KUKA KRL program: ab_com_01_st01_g01.src, ab_com_01_st01_g01.dat

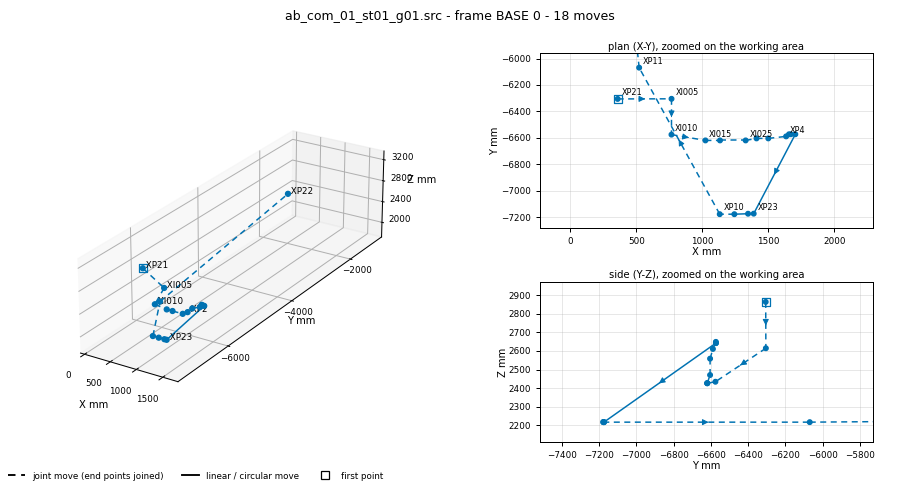
[picture p0: tool path of ab_com_01_st01_g01.src in frame BASE 0, 18 of 18 moves have a stored position in this frame; points joined in program order, loops and branches not executed]
--- ab_com_01_st01_g01.src ---
&ACCESS RVP
&REL 140
&COMMENT Dep Travessa axor atego
&PARAM DISKPATH = KRC:\R1\Program\OLP
&PARAM TEMPLATE = C:\KRC\Roboter\Template\vorgabe
&PARAM EDITMASK = *
DEF ab_com_01_st01_g01( )
;FOLD INI
  ;FOLD BASISTECH INI
    GLOBAL INTERRUPT DECL 3 WHEN $STOPMESS==TRUE DO IR_STOPM ( )
    INTERRUPT ON 3
    BAS (#INITMOV,0)
  ;ENDFOLD (BASISTECH INI)
;FOLD GRIPPERTECH INI
USER_GRP(0,DUMMY,DUMMY,GDEFAULT)
;ENDFOLD (GRIPPERTECH INI)
  ;FOLD USER INI
    ;Make your modifications here

  ;ENDFOLD (USER INI)
;ENDFOLD (INI)

; Caracterizacao dos meios de producao
; Changes: Deposita LCA na GeoBox
; Modelos: Axor/Atego - ETB/LTA/LTB/STB
; Versao Atual: 31/03/2016
; Name: P13.050-R2

chk_w7_wechs_ok( )     ; CHECK GRIPPER AXOR/ATEGO

;FOLD PTP P21 CONT Vel=100 % PDAT15 Tool[7]:Garra AXOR Base[0];%{PE}%R 8.2.20,%MKUKATPBASIS,%CMOVE,%VPTP,%P 1:PTP, 2:P21, 3:C_DIS, 5:100, 7:PDAT15
$BWDSTART=FALSE
PDAT_ACT=PPDAT15
FDAT_ACT=FP21
BAS(#PTP_PARAMS,100)
PTP XP21 C_DIS
;ENDFOLD

; ABRE GRAMPOS E VERIFICA
;FOLD SET Z2.1 RPS AXOR State=OPN CONT at START Delay=1 ms;%{PE}%R 8.2.1,%MKUKATPGRP,%CGRP,%VGRP,%P 2:10, 4:1, 5:#YES, 6:GDAT17, 8:0, 10:1
TRIGGER WHEN DISTANCE=0 DELAY=1 DO H50(GRP_APO,10,1,GCONT) PRIO=-1
;ENDFOLD
;FOLD SET Z3.1 GRP AXOR State=OPN CONT at START Delay=1 ms;%{PE}%R 8.2.1,%MKUKATPGRP,%CGRP,%VGRP,%P 2:11, 4:1, 5:#YES, 6:GDAT18, 8:0, 10:1
TRIGGER WHEN DISTANCE=0 DELAY=1 DO H50(GRP_APO,11,1,GCONT) PRIO=-1
;ENDFOLD
;FOLD SET Z5.1/2/3/4 GRP AXOR State=OPN CONT at START Delay=1 ms;%{PE}%R 8.2.1,%MKUKATPGRP,%CGRP,%VGRP,%P 2:13, 4:1, 5:#YES, 6:GDAT20, 8:0, 10:1
TRIGGER WHEN DISTANCE=0 DELAY=1 DO H50(GRP_APO,13,1,GCONT) PRIO=-1
;ENDFOLD
;FOLD SET Z6.1/2/3/4 GRP AXOR State=OPN CONT at START Delay=1 ms;%{PE}%R 8.2.1,%MKUKATPGRP,%CGRP,%VGRP,%P 2:14, 4:1, 5:#YES, 6:GDAT21, 8:0, 10:1
TRIGGER WHEN DISTANCE=0 DELAY=1 DO H50(GRP_APO,14,1,GCONT) PRIO=-1
;ENDFOLD
;FOLD SET Z7.1/2 GRP AXOR State=OPN GDAT24;%{PE}%R 8.2.1,%MKUKATPGRP,%CGRP,%VGRP,%P 2:15, 4:1, 5:#NO, 6:GDAT24, 8:0, 10:1
H50(GRP,15,1,GGDAT24)
;ENDFOLD
chk_w7_rps2_opn()
chk_w7_grp3_opn()
chk_w7_grp5_opn()
chk_w7_grp6_opn()
chk_w7_grp7_opn()

;FOLD OUT 3374 'Lib. Dep. Axor/Atego' State=TRUE ;%{PE}%R 8.2.20,%MKUKATPBASIS,%COUT,%VOUTX,%P 2:3374, 3:Lib. Dep. Axor/Atego, 5:TRUE, 6:
$OUT[3374]=TRUE
;ENDFOLD
;FOLD WAIT FOR ( IN 3374 'Lib. Deposito Axor/Atego' );%{PE}%R 8.2.20,%MKUKATPBASIS,%CEXT_WAIT_FOR,%VEXT_WAIT_FOR,%P 2:, 4:, 5:$IN, 6:3374, 7:Lib. Deposito Axor/Atego, 9:
WAIT FOR  ( $IN[3374] )
;ENDFOLD
;FOLD OUT 3374 'Lib. Dep. Axor/Atego' State=FALSE ;%{PE}%R 8.2.20,%MKUKATPBASIS,%COUT,%VOUTX,%P 2:3374, 3:Lib. Dep. Axor/Atego, 5:FALSE, 6:
$OUT[3374]=FALSE
;ENDFOLD

;FOLD PTP l005 CONT Vel=100 % P_OLP2 Tool[7]:Garra AXOR Base[0];%{PE}%R 8.2.20,%MKUKATPBASIS,%CMOVE,%VPTP,%P 1:PTP, 2:l005, 3:C_DIS, 5:100, 7:P_OLP2
$BWDSTART=FALSE
PDAT_ACT=PP_OLP2
FDAT_ACT=Fl005
BAS(#PTP_PARAMS,100)
PTP Xl005 C_DIS
;ENDFOLD
;FOLD PTP l010 CONT Vel=100 % P_OLP3 Tool[7]:Garra AXOR Base[0];%{PE}%R 8.2.20,%MKUKATPBASIS,%CMOVE,%VPTP,%P 1:PTP, 2:l010, 3:C_DIS, 5:100, 7:P_OLP3
$BWDSTART=FALSE
PDAT_ACT=PP_OLP3
FDAT_ACT=Fl010
BAS(#PTP_PARAMS,100)
PTP Xl010 C_DIS
;ENDFOLD

; LIGA INTERTRAVAMENTO 5 C/ R5 GARRA
;FOLD Collision.Monitoring_5_On ;%{PE}%MKUKATPUSER
COLLSTOP( 5, 1 ) ;not Interrupt-Controlled
;ENDFOLD

;FOLD ; ABRE GRAMPO Z4.1 "LCA";%{PE}%R 8.2.20,%MKUKATPBASIS,%CCOMMENT,%VNORMAL,%P 2:ABRE  GRAMPO  Z4.1  "LCA"
;ENDFOLD
;FOLD SET Z4.1 GRP AXOR State=OPN CONT at START Delay=1 ms;%{PE}%R 8.2.1,%MKUKATPGRP,%CGRP,%VGRP,%P 2:12, 4:1, 5:#YES, 6:GDAT4, 8:0, 10:1
TRIGGER WHEN DISTANCE=0 DELAY=1 DO H50(GRP_APO,12,1,GCONT) PRIO=-1
;ENDFOLD

;FOLD PTP l015 CONT Vel=100 % P_OLP4 Tool[7]:Garra AXOR Base[0];%{PE}%R 8.2.20,%MKUKATPBASIS,%CMOVE,%VPTP,%P 1:PTP, 2:l015, 3:C_DIS, 5:100, 7:P_OLP4
$BWDSTART=FALSE
PDAT_ACT=PP_OLP4
FDAT_ACT=Fl015
BAS(#PTP_PARAMS,100)
PTP Xl015 C_DIS
;ENDFOLD
;FOLD PTP l020 CONT Vel=100 % P_OLP5 Tool[7]:Garra AXOR Base[0];%{PE}%R 8.2.20,%MKUKATPBASIS,%CMOVE,%VPTP,%P 1:PTP, 2:l020, 3:C_DIS, 5:100, 7:P_OLP5
$BWDSTART=FALSE
PDAT_ACT=PP_OLP5
FDAT_ACT=Fl020
BAS(#PTP_PARAMS,100)
PTP Xl020 C_DIS
;ENDFOLD
;FOLD PTP l025 CONT Vel=100 % P_OLP6 Tool[7]:Garra AXOR Base[0];%{PE}%R 8.2.20,%MKUKATPBASIS,%CMOVE,%VPTP,%P 1:PTP, 2:l025, 3:C_DIS, 5:100, 7:P_OLP6
$BWDSTART=FALSE
PDAT_ACT=PP_OLP6
FDAT_ACT=Fl025
BAS(#PTP_PARAMS,100)
PTP Xl025 C_DIS
;ENDFOLD
;FOLD PTP P2 CONT Vel=100 % PDAT2 Tool[7]:Garra AXOR Base[0];%{PE}%R 8.2.20,%MKUKATPBASIS,%CMOVE,%VPTP,%P 1:PTP, 2:P2, 3:C_DIS, 5:100, 7:PDAT2
$BWDSTART=FALSE
PDAT_ACT=PPDAT2
FDAT_ACT=FP2
BAS(#PTP_PARAMS,100)
PTP XP2 C_DIS
;ENDFOLD



;FOLD PTP P3 CONT Vel=100 % PDAT3 Tool[7]:Garra AXOR Base[0];%{PE}%R 8.2.20,%MKUKATPBASIS,%CMOVE,%VPTP,%P 1:PTP, 2:P3, 3:C_DIS, 5:100, 7:PDAT3
$BWDSTART=FALSE
PDAT_ACT=PPDAT3
FDAT_ACT=FP3
BAS(#PTP_PARAMS,100)
PTP XP3 C_DIS
;ENDFOLD
;FOLD PTP P4 CONT Vel=100 % PDAT4 Tool[7]:Garra AXOR Base[0];%{PE}%R 8.2.20,%MKUKATPBASIS,%CMOVE,%VPTP,%P 1:PTP, 2:P4, 3:C_DIS, 5:100, 7:PDAT4
$BWDSTART=FALSE
PDAT_ACT=PPDAT4
FDAT_ACT=FP4
BAS(#PTP_PARAMS,100)
PTP XP4 C_DIS
;ENDFOLD
;FOLD PTP P5 CONT Vel=100 % PDAT5 Tool[7]:Garra AXOR Base[0];%{PE}%R 8.2.20,%MKUKATPBASIS,%CMOVE,%VPTP,%P 1:PTP, 2:P5, 3:C_DIS, 5:100, 7:PDAT5
$BWDSTART=FALSE
PDAT_ACT=PPDAT5
FDAT_ACT=FP5
BAS(#PTP_PARAMS,100)
PTP XP5 C_DIS
;ENDFOLD
;FOLD LIN P_DE07 Vel=0.5 m/s L_OLP3 Tool[7]:Garra AXOR Base[0];%{PE}%R 8.2.20,%MKUKATPBASIS,%CMOVE,%VLIN,%P 1:LIN, 2:P_DE07, 3:, 5:0.5, 7:L_OLP3
$BWDSTART=FALSE
LDAT_ACT=LL_OLP3
FDAT_ACT=FP_DE07
BAS(#CP_PARAMS,0.5)
LIN XP_DE07
;ENDFOLD

; VERIFICA PRESENCA LCA
IF (NOT(GHOST())) THEN
;FOLD WAIT FOR ( IN 489 'Presença pç 1 - Axor LCA' );%{PE}%R 8.2.20,%MKUKATPBASIS,%CEXT_WAIT_FOR,%VEXT_WAIT_FOR,%P 2:, 4:, 5:$IN, 6:489, 7:Presença pç 1 - Axor LCA, 9:
WAIT FOR  ( $IN[489] )
;ENDFOLD
ENDIF

;FOLD ; VERIFICA GRAMPO Z4.1 ABERTO "LCA";%{PE}%R 8.2.20,%MKUKATPBASIS,%CCOMMENT,%VNORMAL,%P 2:VERIFICA  GRAMPO  Z4.1  ABERTO  "LCA"
;ENDFOLD
chk_w7_grp4_opn()

;FOLD ; POSICAO DE DEPOSITO;%{PE}%R 8.2.20,%MKUKATPBASIS,%CCOMMENT,%VNORMAL,%P 2:POSICAO  DE  DEPOSITO
;ENDFOLD
;FOLD LIN l030 Vel=0.25 m/s L_OLP2 Tool[7]:Garra AXOR Base[0];%{PE}%R 8.2.20,%MKUKATPBASIS,%CMOVE,%VLIN,%P 1:LIN, 2:l030, 3:, 5:0.25, 7:L_OLP2
$BWDSTART=FALSE
LDAT_ACT=LL_OLP2
FDAT_ACT=Fl030
BAS(#CP_PARAMS,0.25)
LIN Xl030
;ENDFOLD

IF (NOT(GHOST())) THEN
;FOLD WAIT FOR ( IN 490 'Presença pç 2 - Axor Coluna B' ) AND ( IN 491 'Presença pç 3 - Axor Inferior' ) AND ( IN 492 'Presença pç 2 - Axor Coluna A' );%{PE}%R 8.2.20,%MKUKATPBASIS,%CEXT_WAIT_FOR,%VEXT_WAIT_FOR,%P 2:, 4:, 5:$IN, 6:490, 7:Presença pç 2 - Axor Coluna B, 9:AND, 10:, 12:, 13:$IN, 14:491, 15:Presença pç 3 - Axor Inferior, 17:AND, 18:, 20:, 21:$IN, 22:492, 23:Presença pç 2 - Axor Coluna A, 25:
WAIT FOR  ( $IN[490] ) AND ( $IN[491] ) AND ( $IN[492] )
;ENDFOLD
ENDIF

;FOLD OUT 3375 'Lib. p/ sair s/ Gripper Axor/Atego' State=TRUE ;%{PE}%R 8.2.20,%MKUKATPBASIS,%COUT,%VOUTX,%P 2:3375, 3:Lib. p/ sair s/ Gripper Axor/Atego, 5:TRUE, 6:
$OUT[3375]=TRUE
;ENDFOLD

; FECHA GRAMPOS
;FOLD SET Z2.1 RPS AXOR State=CLO GDAT8;%{PE}%R 8.2.1,%MKUKATPGRP,%CGRP,%VGRP,%P 2:10, 4:2, 5:#NO, 6:GDAT8, 8:0, 10:0
H50(GRP,10,2,GGDAT8)
;ENDFOLD
;FOLD SET Z3.1 GRP AXOR State=CLO GDAT9;%{PE}%R 8.2.1,%MKUKATPGRP,%CGRP,%VGRP,%P 2:11, 4:2, 5:#NO, 6:GDAT9, 8:0, 10:0
H50(GRP,11,2,GGDAT9)
;ENDFOLD
;FOLD SET Z5.1/2/3/4 GRP AXOR State=CLO GDAT11;%{PE}%R 8.2.1,%MKUKATPGRP,%CGRP,%VGRP,%P 2:13, 4:2, 5:#NO, 6:GDAT11, 8:0, 10:0
H50(GRP,13,2,GGDAT11)
;ENDFOLD
;FOLD SET Z6.1/2/3/4 GRP AXOR State=CLO GDAT12;%{PE}%R 8.2.1,%MKUKATPGRP,%CGRP,%VGRP,%P 2:14, 4:2, 5:#NO, 6:GDAT12, 8:0, 10:0
H50(GRP,14,2,GGDAT12)
;ENDFOLD

; VERIFICA GRAMPOS FECHADOS
chk_w7_rps2_clo()
chk_w7_grp3_clo()

; FECHA GRAMPO Z4.1
;FOLD SET Z4.1 GRP AXOR State=CLO GDAT14;%{PE}%R 8.2.1,%MKUKATPGRP,%CGRP,%VGRP,%P 2:12, 4:2, 5:#NO, 6:GDAT14, 8:0, 10:0
H50(GRP,12,2,GGDAT14)
;ENDFOLD
;FOLD SET Z7.1/2 GRP AXOR State=CLO GDAT23;%{PE}%R 8.2.1,%MKUKATPGRP,%CGRP,%VGRP,%P 2:15, 4:2, 5:#NO, 6:GDAT23, 8:0, 10:0
H50(GRP,15,2,GGDAT23)
;ENDFOLD

; VERIFICA GRAMPOS FECHADOS
chk_w7_grp5_clo()
chk_w7_grp6_clo()
chk_w7_grp7_clo()
chk_w7_grp4_clo()

; DESLIGA VACUO e VERIFICA
;FOLD SET VACUO AXOR State=BLOW GDAT15;%{PE}%R 8.2.1,%MKUKATPGRP,%CGRP,%VGRP,%P 2:9, 4:2, 5:#NO, 6:GDAT15, 8:0, 10:0
H50(GRP,9,2,GGDAT15)
;ENDFOLD
;FOLD SET VACUO AXOR State=OFF GDAT16;%{PE}%R 8.2.1,%MKUKATPGRP,%CGRP,%VGRP,%P 2:9, 4:3, 5:#NO, 6:GDAT16, 8:0, 10:0
H50(GRP,9,3,GGDAT16)
;ENDFOLD
chk_w7_grp1_vacoff()

; VERIFICA PRESENCA LCA
IF (NOT(GHOST())) THEN
;FOLD WAIT FOR ( IN 489 'Presença pç 1 - Axor LCA' );%{PE}%R 8.2.20,%MKUKATPBASIS,%CEXT_WAIT_FOR,%VEXT_WAIT_FOR,%P 2:, 4:, 5:$IN, 6:489, 7:Presença pç 1 - Axor LCA, 9:
WAIT FOR  ( $IN[489] )
;ENDFOLD
ENDIF

;FOLD OUT 3375 'Lib. p/ sair s/ Gripper Axor/Atego' State=TRUE ;%{PE}%R 8.2.20,%MKUKATPBASIS,%COUT,%VOUTX,%P 2:3375, 3:Lib. p/ sair s/ Gripper Axor/Atego, 5:TRUE, 6:
$OUT[3375]=TRUE
;ENDFOLD
;FOLD WAIT FOR ( IN 3375 'Lib. p/ sair s/ Gripper Axor/Atego' );%{PE}%R 8.2.20,%MKUKATPBASIS,%CEXT_WAIT_FOR,%VEXT_WAIT_FOR,%P 2:, 4:, 5:$IN, 6:3375, 7:Lib. p/ sair s/ Gripper Axor/Atego, 9:
WAIT FOR  ( $IN[3375] )
;ENDFOLD
;FOLD OUT 3375 'Lib. p/ sair s/ Gripper Axor/Atego' State=FALSE ;%{PE}%R 8.2.20,%MKUKATPBASIS,%COUT,%VOUTX,%P 2:3375, 3:Lib. p/ sair s/ Gripper Axor/Atego, 5:FALSE, 6:
$OUT[3375]=FALSE
;ENDFOLD

;FOLD IBUS OFF;%{PE}%R 8.2.20,%MKUKATPBASIS,%CIBUS,%VMAP,%P 2:#OFF, 3:1
$IBUS_OFF=$IBUS_ON
$IBUS_ON=0
;ENDFOLD
;FOLD WAIT Time=0.15 sec;%{PE}%R 8.2.20,%MKUKATPBASIS,%CWAIT,%VWAIT,%P 3:0.15
WAIT SEC 0.15
;ENDFOLD
;FOLD OUT 224 'Bloquear MPS' State=FALSE ;%{PE}%R 8.2.20,%MKUKATPBASIS,%COUT,%VOUTX,%P 2:224, 3:Bloquear MPS, 5:FALSE, 6:
$OUT[224]=FALSE
;ENDFOLD
;FOLD OUT 223 'Desbloquear MPS' State=TRUE ;%{PE}%R 8.2.20,%MKUKATPBASIS,%COUT,%VOUTX,%P 2:223, 3:Desbloquear MPS, 5:TRUE, 6:
$OUT[223]=TRUE
;ENDFOLD
;FOLD WAIT FOR ( IN 217 'MPS Destravado' );%{PE}%R 8.2.20,%MKUKATPBASIS,%CEXT_WAIT_FOR,%VEXT_WAIT_FOR,%P 2:, 4:, 5:$IN, 6:217, 7:MPS Destravado, 9:
WAIT FOR  ( $IN[217] )
;ENDFOLD
;FOLD WAIT FOR NOT ( IN 221 'MPS Travado' );%{PE}%R 8.2.20,%MKUKATPBASIS,%CEXT_WAIT_FOR,%VEXT_WAIT_FOR,%P 2:NOT, 4:, 5:$IN, 6:221, 7:MPS Travado, 9:
WAIT FOR  NOT ( $IN[221] )
;ENDFOLD

;FOLD LIN P23 Vel=0.25 m/s CPDAT9 Tool[8]:Tool Changer Base[0];%{PE}%R 8.2.20,%MKUKATPBASIS,%CMOVE,%VLIN,%P 1:LIN, 2:P23, 3:, 5:0.25, 7:CPDAT9
$BWDSTART=FALSE
LDAT_ACT=LCPDAT9
FDAT_ACT=FP23
BAS(#CP_PARAMS,0.25)
LIN XP23
;ENDFOLD

;FOLD WAIT FOR NOT ( IN 219 'Posicao p/ Acoplamento OK' );%{PE}%R 8.2.20,%MKUKATPBASIS,%CEXT_WAIT_FOR,%VEXT_WAIT_FOR,%P 2:NOT, 4:, 5:$IN, 6:219, 7:Posicao p/ Acoplamento OK, 9:
WAIT FOR  NOT ( $IN[219] )
;ENDFOLD

;FOLD LIN P7 Vel=0.25 m/s CPDAT2 Tool[8]:Tool Changer Base[0];%{PE}%R 8.2.20,%MKUKATPBASIS,%CMOVE,%VLIN,%P 1:LIN, 2:P7, 3:, 5:0.25, 7:CPDAT2
$BWDSTART=FALSE
LDAT_ACT=LCPDAT2
FDAT_ACT=FP7
BAS(#CP_PARAMS,0.25)
LIN XP7
;ENDFOLD

; DESLIGA INTERTRAVAMENTO 5 C/ R5 GARRA
;FOLD Collision.Monitoring_5_Off . ;%{PE}%MKUKATPUSER
COLLSTOP( 5, 2+0 )
;ENDFOLD

;FOLD WAIT FOR NOT ( IN 219 'Posicao p/ Acoplamento OK' );%{PE}%R 8.2.20,%MKUKATPBASIS,%CEXT_WAIT_FOR,%VEXT_WAIT_FOR,%P 2:NOT, 4:, 5:$IN, 6:219, 7:Posicao p/ Acoplamento OK, 9:
WAIT FOR  NOT ( $IN[219] )
;ENDFOLD
;FOLD OUT 223 'Desbloquear MPS' State=FALSE ;%{PE}%R 8.2.20,%MKUKATPBASIS,%COUT,%VOUTX,%P 2:223, 3:Desbloquear MPS, 5:FALSE, 6:
$OUT[223]=FALSE
;ENDFOLD

;FOLD LIN P9 CONT Vel=1 m/s CPDAT4 Tool[7]:Garra AXOR Base[0];%{PE}%R 8.2.20,%MKUKATPBASIS,%CMOVE,%VLIN,%P 1:LIN, 2:P9, 3:C_DIS C_DIS, 5:1, 7:CPDAT4
$BWDSTART=FALSE
LDAT_ACT=LCPDAT4
FDAT_ACT=FP9
BAS(#CP_PARAMS,1)
LIN XP9 C_DIS C_DIS
;ENDFOLD
;FOLD PTP P10 CONT Vel=100 % PDAT6 Tool[7]:Garra AXOR Base[0];%{PE}%R 8.2.20,%MKUKATPBASIS,%CMOVE,%VPTP,%P 1:PTP, 2:P10, 3:C_DIS, 5:100, 7:PDAT6
$BWDSTART=FALSE
PDAT_ACT=PPDAT6
FDAT_ACT=FP10
BAS(#PTP_PARAMS,100)
PTP XP10 C_DIS
;ENDFOLD
;FOLD PTP P11 CONT Vel=100 % PDAT7 Tool[7]:Garra AXOR Base[0];%{PE}%R 8.2.20,%MKUKATPBASIS,%CMOVE,%VPTP,%P 1:PTP, 2:P11, 3:C_DIS, 5:100, 7:PDAT7
$BWDSTART=FALSE
PDAT_ACT=PPDAT7
FDAT_ACT=FP11
BAS(#PTP_PARAMS,100)
PTP XP11 C_DIS
;ENDFOLD

;FOLD OUT 3348 'Fora area GEOBOX' State=TRUE ;%{PE}%R 8.2.20,%MKUKATPBASIS,%COUT,%VOUTX,%P 2:3348, 3:Fora area GEOBOX, 5:TRUE, 6:
$OUT[3348]=TRUE
;ENDFOLD
;FOLD PULSE 3343 'R2 entregou peça geo' State=TRUE Time=3 sec;%{PE}%R 8.2.20,%MKUKATPBASIS,%COUT,%VPULSE,%P 2:3343, 3:R2 entregou peça geo, 5:TRUE, 6:, 8:3
PULSE($OUT[3343], TRUE,3)
;ENDFOLD

;FOLD PTP P22 CONT Vel=100 % PDAT16 Tool[7]:Garra AXOR Base[0];%{PE}%R 8.2.20,%MKUKATPBASIS,%CMOVE,%VPTP,%P 1:PTP, 2:P22, 3:C_DIS, 5:100, 7:PDAT16
$BWDSTART=FALSE
PDAT_ACT=PPDAT16
FDAT_ACT=FP22
BAS(#PTP_PARAMS,100)
PTP XP22 C_DIS
;ENDFOLD

END

--- ab_com_01_st01_g01.dat ---
&ACCESS RVP
&REL 140
&COMMENT Dep Travessa axor atego
&PARAM DISKPATH = KRC:\R1\Program\OLP
&PARAM TEMPLATE = C:\KRC\Roboter\Template\vorgabe
&PARAM EDITMASK = *
DEFDAT  ab_com_01_st01_g01
;FOLD EXTERNAL DECLARATIONS;%{PE}%MKUKATPBASIS,%CEXT,%VCOMMON,%P
;FOLD GRIPPERTECH EXT
EXT  H50 (INT  :IN,INT  :IN,INT  :IN,GRP_TYP  :IN )
;ENDFOLD (GRIPPERTECH EXT)
;FOLD SPOTTECH EXT

;ENDFOLD (SPOTTECH EXT)
;FOLD BASISTECH EXT;%{PE}%MKUKATPBASIS,%CEXT,%VEXT,%P
EXT  BAS (BAS_COMMAND  :IN,REAL  :IN )
DECL INT SUCCESS
;ENDFOLD (BASISTECH EXT)
;FOLD USER EXT;%{E}%MKUKATPUSER,%CEXT,%VEXT,%P
;Make your modifications here

;ENDFOLD (USER EXT)
;ENDFOLD (EXTERNAL DECLARATIONS)
DECL FDAT Fl005={TOOL_NO 7,BASE_NO 0,IPO_FRAME #BASE,POINT2[] " ",TQ_STATE FALSE}
DECL PDAT PP_OLP2={VEL 100.0,ACC 100.0,APO_DIST 50.0,APO_MODE #CDIS}
DECL E6POS Xl005={X 767.053223,Y -6304.99023,Z 2614.30005,A -171.571304,B 67.8797913,C 115.369499,S 6,T 50,E1 -4975.82813,E2 0.0,E3 0.0,E4 0.0,E5 0.0,E6 0.0}
DECL FDAT Fl010={TOOL_NO 7,BASE_NO 0,IPO_FRAME #BASE,POINT2[] " ",TQ_STATE FALSE}
DECL PDAT PP_OLP3={VEL 100.0,ACC 100.0,APO_DIST 30.0,APO_MODE #CDIS}
DECL E6POS Xl010={X 766.797607,Y -6575.89404,Z 2434.36694,A -171.574203,B 67.8798065,C 115.367104,S 6,T 50,E1 -4975.82715,E2 0.0,E3 0.0,E4 0.0,E5 0.0,E6 0.0}
DECL FDAT Fl015={TOOL_NO 7,BASE_NO 0,IPO_FRAME #BASE,POINT2[] " ",TQ_STATE FALSE}
DECL PDAT PP_OLP4={VEL 100.0,ACC 100.0,APO_DIST 50.0,APO_MODE #CDIS}
DECL E6POS Xl015={X 1023.69598,Y -6619.8418,Z 2426.50708,A -178.543701,B 68.1228333,C 107.851097,S 6,T 51,E1 -4975.82813,E2 0.0,E3 0.0,E4 0.0,E5 0.0,E6 0.0}
DECL FDAT Fl020={TOOL_NO 7,BASE_NO 0,IPO_FRAME #BASE,POINT2[] " ",TQ_STATE FALSE}
DECL PDAT PP_OLP5={VEL 100.0,ACC 100.0,APO_DIST 50.0,APO_MODE #CDIS}
DECL E6POS Xl020={X 1133.97998,Y -6619.84521,Z 2426.5061,A -178.544205,B 68.1227798,C 107.8507,S 6,T 51,E1 -4975.83008,E2 0.0,E3 0.0,E4 0.0,E5 0.0,E6 0.0}
DECL FDAT Fl025={TOOL_NO 7,BASE_NO 0,IPO_FRAME #BASE,POINT2[] " ",TQ_STATE FALSE}
DECL PDAT PP_OLP6={VEL 100.0,ACC 100.0,APO_DIST 50.0,APO_MODE #CDIS}
DECL E6POS Xl025={X 1327.97595,Y -6619.84521,Z 2426.5061,A -178.544495,B 68.1227264,C 107.850304,S 6,T 51,E1 -4975.8291,E2 0.0,E3 0.0,E4 0.0,E5 0.0,E6 0.0}
DECL FDAT Fl030={TOOL_NO 7,BASE_NO 0,IPO_FRAME #BASE,POINT2[] " ",TQ_STATE FALSE}
DECL E6POS Xl030={X 1704.104,Y -6573.39893,Z 2641.80103,A -17.8527508,B 89.5465927,C -92.7548523,S 6,T 51,E1 -4975.83203,E2 0.0,E3 0.0,E4 0.0,E5 0.0,E6 0.0}
DECL LDAT LL_OLP2={VEL 0.25,ACC 100.0,APO_DIST 0.0,APO_FAC 0.0,ORI_TYP #VAR,CIRC_TYP #BASE,JERK_FAC 50.0}
DECL BASIS_SUGG_T LAST_BASIS={POINT1[] "P0                      ",POINT2[] "P0                      ",CP_PARAMS[] "CPDAT0                  ",PTP_PARAMS[] "PDAT0                   ",CONT[] "                        ",CP_VEL[] "0.25                    ",PTP_VEL[] "100                     ",SYNC_PARAMS[] "SYNCDAT                 ",SPL_NAME[] "S0                      "}
DECL E6POS XP2={X 1410.349,Y -6604.56494,Z 2470.51392,A -178.043396,B 75.4370193,C 108.513298,S 6,T 51,E1 -4975.83008,E2 0.0,E3 0.0,E4 0.0,E5 0.0,E6 0.0}
DECL FDAT FP2={TOOL_NO 7,BASE_NO 0,IPO_FRAME #BASE,POINT2[] " ",TQ_STATE FALSE}
DECL PDAT PPDAT2={VEL 100.0,ACC 100.0,APO_DIST 50.0,APO_MODE #CDIS}
DECL E6POS XP3={X 1499.45703,Y -6604.54688,Z 2558.42505,A -176.547699,B 81.7896729,C 110.035797,S 6,T 51,E1 -4975.83008,E2 0.0,E3 0.0,E4 0.0,E5 0.0,E6 0.0}
DECL FDAT FP3={TOOL_NO 7,BASE_NO 0,IPO_FRAME #BASE,POINT2[] " ",TQ_STATE FALSE}
DECL PDAT PPDAT3={VEL 100.0,ACC 100.0,APO_DIST 50.0,APO_MODE #CDIS}
DECL E6POS XP4={X 1634.35303,Y -6589.39697,Z 2610.59692,A -167.308899,B 87.754921,C 119.300003,S 6,T 51,E1 -4975.8291,E2 0.0,E3 0.0,E4 0.0,E5 0.0,E6 0.0}
DECL FDAT FP4={TOOL_NO 7,BASE_NO 0,IPO_FRAME #BASE,POINT2[] " ",TQ_STATE FALSE}
DECL PDAT PPDAT4={VEL 100.0,ACC 100.0,APO_DIST 50.0,APO_MODE #CDIS}
DECL E6POS XP5={X 1656.11804,Y -6573.39893,Z 2648.57007,A -17.87043,B 89.5466309,C -92.7723999,S 6,T 51,E1 -4975.83301,E2 0.0,E3 0.0,E4 0.0,E5 0.0,E6 0.0}
DECL FDAT FP5={TOOL_NO 7,BASE_NO 0,IPO_FRAME #BASE,POINT2[] " ",TQ_STATE FALSE}
DECL PDAT PPDAT5={VEL 100.0,ACC 100.0,APO_DIST 50.0,APO_MODE #CDIS}
DECL LDAT LL_OLP3={VEL 0.25,ACC 100.0,APO_DIST 0.0,APO_FAC 0.0,ORI_TYP #VAR,CIRC_TYP #BASE,JERK_FAC 50.0}
DECL E6POS XP_DE07={X 1670.52295,Y -6573.39697,Z 2641.79199,A -17.9401093,B 89.5467224,C -92.8419113,S 6,T 51,E1 -4975.83203,E2 0.0,E3 0.0,E4 0.0,E5 0.0,E6 0.0}
DECL FDAT FP_DE07={TOOL_NO 7,BASE_NO 0,IPO_FRAME #BASE,POINT2[] " ",TQ_STATE FALSE}
DECL E6POS XP7={X 1346.37903,Y -7174.67676,Z 2216.93311,A 90.3285828,B -44.8586502,C 89.3926926,S 6,T 51,E1 -4975.8418,E2 0.0,E3 0.0,E4 0.0,E5 0.0,E6 0.0}
DECL FDAT FP7={TOOL_NO 8,BASE_NO 0,IPO_FRAME #BASE,POINT2[] " ",TQ_STATE FALSE}
DECL LDAT LCPDAT2={VEL 2.0,ACC 100.0,APO_DIST 100.0,APO_FAC 50.0,AXIS_VEL 100.0,AXIS_ACC 100.0,ORI_TYP #VAR,CIRC_TYP #BASE,JERK_FAC 50.0,GEAR_JERK 50.0,EXAX_IGN 0}
DECL E6POS XP9={X 1242.55298,Y -7178.2959,Z 2218.17212,A 90.328598,B -44.8586502,C 89.3926773,S 6,T 51,E1 -4975.8418,E2 0.0,E3 0.0,E4 0.0,E5 0.0,E6 0.0}
DECL FDAT FP9={TOOL_NO 8,BASE_NO 0,IPO_FRAME #BASE,POINT2[] " ",TQ_STATE FALSE}
DECL LDAT LCPDAT4={VEL 2.0,ACC 100.0,APO_DIST 100.0,APO_FAC 50.0,AXIS_VEL 100.0,AXIS_ACC 100.0,ORI_TYP #VAR,CIRC_TYP #BASE,JERK_FAC 50.0,GEAR_JERK 50.0,EXAX_IGN 0}
DECL E6POS XP10={X 1131.93701,Y -7178.10303,Z 2217.34106,A 90.328598,B -44.8586502,C 89.3926773,S 6,T 51,E1 -4975.8418,E2 0.0,E3 0.0,E4 0.0,E5 0.0,E6 0.0}
DECL FDAT FP10={TOOL_NO 8,BASE_NO 0,IPO_FRAME #BASE,POINT2[] " ",TQ_STATE FALSE}
DECL PDAT PPDAT6={VEL 100.0,ACC 100.0,APO_DIST 100.0,APO_MODE #CDIS}
DECL GRP_SUGG_T LAST_GRP={NUMBER[] "9                       ",STATE[] "3                       ",PARAMS[] "GDAT16                  "}
DECL GRP_TYP GGDAT1={G_APO #NO,GRP_TIME 0.200000003,CTRL #OFF,DLY 0,DST 1}
DECL GRP_TYP GGDAT2={G_APO #NO,GRP_TIME 0.200000003,CTRL #OFF,DLY 0,DST 1}
DECL GRP_TYP GGDAT3={G_APO #NO,GRP_TIME 0.200000003,CTRL #OFF,DLY 0,DST 1}
DECL GRP_TYP GGDAT4={G_APO #NO,GRP_TIME 0.200000003,CTRL #OFF,DLY 0,DST 1}
DECL GRP_TYP GGDAT5={G_APO #NO,GRP_TIME 0.200000003,CTRL #OFF,DLY 0,DST 1}
DECL GRP_TYP GGDAT6={G_APO #NO,GRP_TIME 0.200000003,CTRL #OFF,DLY 0,DST 1}
DECL GRP_TYP GGDAT7={G_APO #NO,GRP_TIME 0.200000003,CTRL #OFF,DLY 0,DST 1}
DECL GRP_TYP GGDAT8={G_APO #NO,GRP_TIME 0.200000003,CTRL #OFF,DLY 0,DST 1}
DECL GRP_TYP GGDAT9={G_APO #NO,GRP_TIME 0.200000003,CTRL #OFF,DLY 0,DST 1}
DECL GRP_TYP GGDAT10={G_APO #NO,GRP_TIME 0.200000003,CTRL #OFF,DLY 0,DST 1}
DECL GRP_TYP GGDAT11={G_APO #NO,GRP_TIME 0.200000003,CTRL #OFF,DLY 0,DST 1}
DECL GRP_TYP GGDAT12={G_APO #NO,GRP_TIME 0.200000003,CTRL #OFF,DLY 0,DST 1}
DECL GRP_TYP GGDAT13={G_APO #NO,GRP_TIME 0.200000003,CTRL #OFF,DLY 0,DST 1}
DECL GRP_TYP GGDAT14={G_APO #NO,GRP_TIME 0.200000003,CTRL #OFF,DLY 0,DST 1}
DECL E6POS XP11={X 522.150879,Y -6069.32617,Z 2217.34302,A 86.9205399,B -44.8586388,C 89.3926468,S 6,T 51,E1 -3832.06909,E2 0.0,E3 0.0,E4 0.0,E5 0.0,E6 0.0}
DECL FDAT FP11={TOOL_NO 8,BASE_NO 0,IPO_FRAME #BASE,POINT2[] " ",TQ_STATE FALSE}
DECL PDAT PPDAT7={VEL 100.0,ACC 100.0,APO_DIST 100.0,APO_MODE #CDIS}
DECL GRP_TYP GGDAT15={G_APO #NO,GRP_TIME 0.200000003,CTRL #OFF,DLY 0,DST 1}
DECL GRP_TYP GGDAT16={G_APO #NO,GRP_TIME 0.200000003,CTRL #OFF,DLY 0,DST 1}
DECL GRP_TYP GGDAT17={G_APO #NO,GRP_TIME 0.200000003,CTRL #OFF,DLY 0,DST 1}
DECL GRP_TYP GGDAT18={G_APO #NO,GRP_TIME 0.200000003,CTRL #OFF,DLY 0,DST 1}
DECL GRP_TYP GGDAT19={G_APO #NO,GRP_TIME 0.200000003,CTRL #OFF,DLY 0,DST 1}
DECL GRP_TYP GGDAT20={G_APO #NO,GRP_TIME 0.200000003,CTRL #OFF,DLY 0,DST 1}
DECL GRP_TYP GGDAT21={G_APO #NO,GRP_TIME 0.200000003,CTRL #OFF,DLY 0,DST 1}
DECL GRP_TYP GGDAT22={G_APO #NO,GRP_TIME 0.200000003,CTRL #OFF,DLY 0,DST 1}
DECL E6POS XP21={X 359.519592,Y -6305.7959,Z 2863.20508,A -161.416397,B 80.027832,C 125.875397,S 6,T 50,E1 -4975.82617,E2 0.0,E3 0.0,E4 0.0,E5 0.0,E6 0.0}
DECL FDAT FP21={TOOL_NO 7,BASE_NO 0,IPO_FRAME #BASE,POINT2[] " ",TQ_STATE FALSE}
DECL PDAT PPDAT15={VEL 100.0,ACC 100.0,APO_DIST 100.0,APO_MODE #CDIS}
DECL E6POS XP22={X 0.000957950426,Y -1148.60498,Z 2255.92505,A 103.8032,B 19.4667301,C -175.319504,S 2,T 10,E1 200.000198,E2 0.0,E3 0.0,E4 0.0,E5 0.0,E6 0.0}
DECL FDAT FP22={TOOL_NO 8,BASE_NO 0,IPO_FRAME #BASE,POINT2[] " ",TQ_STATE FALSE}
DECL PDAT PPDAT16={VEL 100.0,ACC 100.0,APO_DIST 100.0,APO_MODE #CDIS}
DECL E6POS XP23={X 1389.01697,Y -7174.19287,Z 2217.76489,A 90.3317337,B -44.8595581,C 89.3912888,S 6,T 51,E1 -4975.83301,E2 0.0,E3 0.0,E4 0.0,E5 0.0,E6 0.0}
DECL FDAT FP23={TOOL_NO 8,BASE_NO 0,IPO_FRAME #BASE,POINT2[] " ",TQ_STATE FALSE}
DECL LDAT LCPDAT9={VEL 2.0,ACC 100.0,APO_DIST 100.0,APO_FAC 50.0,AXIS_VEL 100.0,AXIS_ACC 100.0,ORI_TYP #VAR,CIRC_TYP #BASE,JERK_FAC 50.0,GEAR_JERK 50.0,EXAX_IGN 0}
DECL GRP_TYP GCONT={G_APO #YES,GRP_TIME 0.0,CTRL #OFF,DLY 0,DST 0}
DECL GRP_TYP GGDAT23={G_APO #NO,GRP_TIME 0.200000003,CTRL #OFF,DLY 0,DST 1}
DECL GRP_TYP GGDAT24={G_APO #NO,GRP_TIME 0.200000003,CTRL #OFF,DLY 0,DST 1}
ENDDAT
